// Mitsubishi GX Works2 project: New circuit plc   PLC: FX1N/FX1NC

PROGRAM MAIN
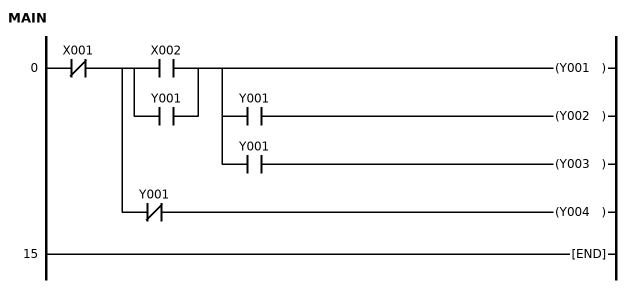
0     LDI     X001
      MPS
      LD      X002
      OR      Y001
      ANB
      OUT     Y001
      MPS
      AND     Y001
      OUT     Y002
      MPP
      AND     Y001
      OUT     Y003
      MPP
      ANI     Y001
      OUT     Y004
15    END
END_PROGRAM
